PROGRAM MAIN
VAR
	fbMotor			:FB_M;
	fbValve			:FB_S;
END_VAR

fbMotor();
fbValve	();

END_PROGRAM

(* stored: Version 1.1.0.1, ProductVersion 3.1.4024.12
   POU MAIN: Id {ab4dde46-4af9-4f37-baaf-4f46d01c1d2e}, SpecialFunc None *)
